% RSLogix 500 project I2P JOB 8.RSS, saved by version 10.00.00.00 %
PROJECT "UNTITLED"    % processor: Bul.1763 MicroLogix 1100 Series B %

PROGRAM FILES
  LAD 2   4 rungs

DATA FILES
  O0 OUTPUT  4 elements
  I1 INPUT  6 elements
  S2 STATUS  66 elements
  B3 BINARY  1 elements
  T4 TIMER  1 elements
  C5 COUNTER  1 elements
  R6 CONTROL  1 elements
  N7 INTEGER  1 elements
  F8 FLOAT  1 elements

LADDER 2
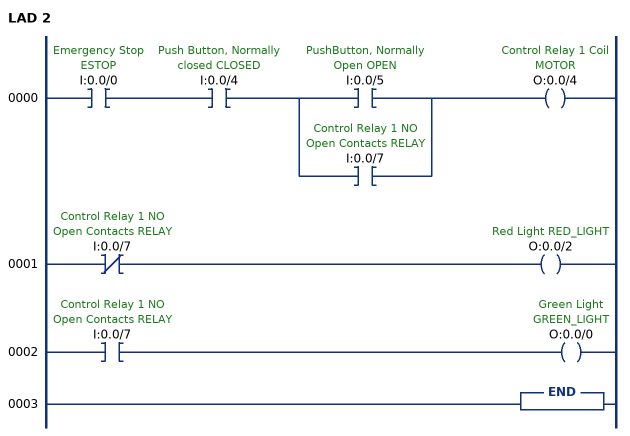
% Rung: 0 %
SOR XIC I:0.0/0 XIC I:0.0/4 BST XIC I:0.0/5 NXB XIC I:0.0/7 BND OTE O:0.0/4 EOR
%   I:0.0/0  ESTOP  "Emergency Stop" %
%   I:0.0/4  CLOSED  "Push Button, Normally closed" %
%   I:0.0/5  OPEN  "PushButton, Normally Open" %
%   I:0.0/7  RELAY  "Control Relay 1 NO Open Contacts" %
%   O:0.0/4  MOTOR  "Control Relay 1 Coil" %
% Rung: 1 %
SOR XIO I:0.0/7 OTE O:0.0/2 EOR
%   I:0.0/7  RELAY  "Control Relay 1 NO Open Contacts" %
%   O:0.0/2  RED_LIGHT  "Red Light" %
% Rung: 2 %
SOR XIC I:0.0/7 OTE O:0.0/0 EOR
%   I:0.0/7  RELAY  "Control Relay 1 NO Open Contacts" %
%   O:0.0/0  GREEN_LIGHT  "Green Light" %
% Rung: 3 %
SOR END EOR

OTHER DOCUMENTED ADDRESSES
  I:0.0/1  FORWARD  "Three Position Selector Switch Position A"
  I:0.0/2  REVERSE  "Three Position Selector Switch, Position B"
  I:0.0/3  "Two Position selector switch"
  I:0.0/6  "PushButton, Normally Open"
